// TwinCAT 3 PLC project cpu
// ProgramVersion: 3.1.4026.1+c9eadab3edd020c56c333d811d5b3c408c2550c8
// libraries:
//   Tc2_Standard, * (Beckhoff Automation GmbH)
//   Tc2_System, * (Beckhoff Automation GmbH)
// project tree:
//   DUTs/ IOpState.TcIO, IValve.TcIO, OpState.TcDUT
//   / MAIN.TcPOU, PlcTask.TcTTO
// real-time tasks:
//   TASK PlcTask: cycle T#10ms, priority 20, ADS port 350

CONFIGURATION cpu
    RESOURCE PLC ON TwinCAT3
        TASK PlcTask(INTERVAL := T#10ms, PRIORITY := 20);
        PROGRAM MAIN WITH PlcTask : MAIN;
    END_RESOURCE
END_CONFIGURATION

// ---- DUTs/OpState.TcDUT
{attribute 'qualified_only'}
{attribute 'strict'}
{attribute 'to_string'}
TYPE OpState :
(
	OP 		:= 0,
	NOT_OP	:= 1
) DINT;
END_TYPE

// ---- DUTs/IOpState.TcIO
INTERFACE IOpState

PROPERTY OpState : OpState
GET
END_GET
END_PROPERTY

END_INTERFACE

// ---- DUTs/IValve.TcIO
INTERFACE IValve

PROPERTY Value : LREAL
GET
END_GET
END_PROPERTY

END_INTERFACE

// ---- MAIN.TcPOU
PROGRAM MAIN
VAR
END_VAR

END_PROGRAM
